(* CODESYS project EZS2_Template.project

Project tree, tasks and I/O mapping:
  Device : Berghof PPC V3 Control, Berghof Automation GmbH, version 3.12.3.0
    application Application
      libraries: Standard, * (System)
      task MainTask (cyclic, interval 4000 µs, priority 16) calls MAIN
      task EtherCAT_Task (cyclic, interval 4000 µs, priority 0) calls EtherCAT_Master.EtherCAT_Task [EtherCAT_Master.EtherCAT_Task]
      global variables Globale_Variablen
      POUs/
        program MAIN [FBD]
        Simulation/
          program SimulationPRG [ST]
          function block SimWerkstueck [SFC]: Init_entry, Einlegestation_active, Band1_active, Uebergabestation1_active, Fraesstation_active, Bohrstation_active, Uebergabestation_active, Ausgabestation_active, Init_active, Init_active_0, Einlegestation_entry
          program Simu [ST]
          function block SimSchieber [ST]
        Steuerung/
          program Steuerung [FBD]
          function block EinAusgabe [SFC]: waitForPstation_entry, bandactive_entry, overshoot_active, overshoot_exit, Init_active, bandactive_active
          function block Uebergabe [SFC]: SationEmty_entry, Push_active, Push_entry, Push_exit, Pull_entry, Pull_active, Pull_exit, StationEmty_exit
      visualisation TAKTSTRASSE
    EtherCAT_Master : EtherCAT Master, 3S - Smart Software Solutions GmbH, version 3.5.8.40
        settings: NetworkName = 'eth1'; NetworkName = "eth1"; SelectNetworkByName = True
      onboard_Buskoppler : onboard Buscoupler, Berghof Automation GmbH, version Revision=16#00000001
          settings: StationAlias = 0; DC sync0 cycletime = 4000; DC sync1 cycletime = 4000
        E_I_O_DI16_DO16 : DI16/DO16 1ms 0.5A (204 800 100), Berghof Automation GmbH, version Revision=16#00000001
            settings: StationAlias = 0; DC sync0 cycletime = 4000; DC sync1 cycletime = 4000
            unmapped channels: DigitalOutput0, DigitalOutput1, DigitalOutput2, DigitalOutput3, DigitalOutput4, DigitalOutput5, DigitalOutput6, DigitalOutput7, DigitalOutput8, DigitalOutput9, DigitalOutput10, DigitalOutput11, DigitalOutput12, DigitalOutput13, DigitalOutput14, DigitalOutput15, DigitalInput0, DigitalInput1, DigitalInput2, DigitalInput3, DigitalInput4, DigitalInput5, DigitalInput6, DigitalInput7, DigitalInput8, DigitalInput9, DigitalInput10, DigitalInput11, DigitalInput12, DigitalInput13, DigitalInput14, DigitalInput15
  libraries: VisuSymbols, 3.5.10.0 (System)
  text list GlobalTextList
*)

// Device/Application/Globale_Variablen
VAR_GLOBAL
(***** STUDENTEN VARIABLEN *****)

	L1:	BOOL;	(* Lichtschranke 1 (Einlegestation) *)
	L2:	BOOL;	(* Lichtschranke 2 (Einlegestation) *)
	L3:	BOOL;	(* Lichtschranke 3 (Fraeser) *)
	L4:	BOOL;	(* Lichtschranke 4 (Bohrer) *)
	L5:	BOOL;	(* Lichtschranke 5 (Ausgabestation) *)
	
	E1:	BOOL;	(* Endtaster 1 (Uebergabestation 1) *)
	E2:	BOOL;	(* Endtaster 2 (Uebergabestation 1) *)
	E3: BOOL;	(* Endtaster 3 (Uebergabestation 2) *)
	E4:	BOOL;	(* Endtaster 4 (Uebergabestation 2) *)
	
	B1	AT %QX0.0:	BOOL;	(* Foerderband 1 (Einlegestation) *)
	B2	AT %QX0.1:	BOOL;	(* Foerderband 2 (Fraeser) *)
	B3	AT %QX0.2:	BOOL;	(* Foerderband 3 (Bohrer) *)
	B4	AT %QX0.3:	BOOL;	(* Foerderband 4 (Ausgabestation) *)
	
	M1	AT %QX0.5:	BOOL;	(* Motor 1 (Uebergabestation 1) *)
	M2	AT %QX0.6:	BOOL;	(* Motor 2 (Fraeser) *)
	M3	AT %QX0.7:	BOOL;	(* Motor 3 (Bohrer) *)
	M4	AT %QX0.8:	BOOL;	(* Motor 4 (Uebergabestation 2) *)
	
	R1	AT %QX0.10:	BOOL;	(* Relais 1 (Uebergabestation 1) *)
	R2	AT %QX0.11:	BOOL;	(* Relais 2 (Uebergabestation 2) *)

(***** ENDE ***** STUDENTEN VARIABLEN *****)

	L1_real	AT %IX0.0:	BOOL;	(* Lichtschranke 1 (Einlegestation) *)
	L2_real	AT %IX0.1:	BOOL;	(* Lichtschranke 2 (Einlegestation) *)
	L3_real	AT %IX0.2:	BOOL;	(* Lichtschranke 3 (Fraeser) *)
	L4_real	AT %IX0.3:	BOOL;	(* Lichtschranke 4 (Bohrer) *)
	L5_real	AT %IX0.4:	BOOL;	(* Lichtschranke 5 (Ausgabestation) *)
	
	E1_real	AT %IX0.6:	BOOL;	(* Endanschlag 1 (Uebergabestation 1) *)
	E2_real	AT %IX0.7:	BOOL;	(* Endanschlag 2 (Uebergabestation 1) *)
	E3_real	AT %IX0.8: 	BOOL;	(* Endanschlag 3 (Uebergabestation 2) *)
	E4_real	AT %IX0.9:	BOOL;	(* Endanschlag 4 (Uebergabestation 2) *)

	SIMULATION: BOOL := TRUE;

END_VAR

// Device/Application/POUs/MAIN
PROGRAM MAIN
VAR
END_VAR

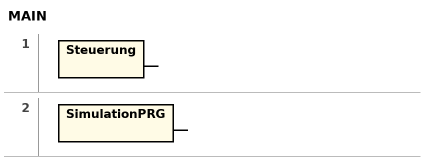
// NETWORK 1
Steuerung();

// NETWORK 2
SimulationPRG();

END_PROGRAM

// Device/Application/POUs/Steuerung/Steuerung
PROGRAM Steuerung
VAR
	Eingabe: EinAusgabe;
	Ue1Emty:BOOL;
	overTimeEin:TIME:=T#2S;
	Uebergabe_1: Uebergabe;
	finishedEin: BOOL;
	toUe1: BOOL;
	toFrae: BOOL;
	Ue1Fin: BOOL;
END_VAR

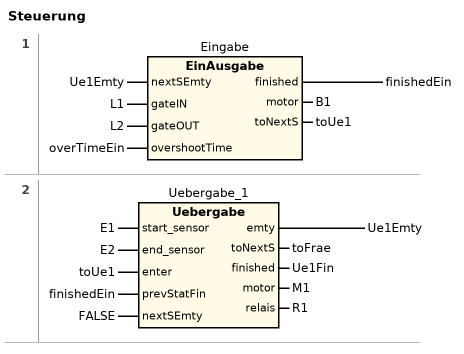
// NETWORK 1
Eingabe(
    nextSEmty := Ue1Emty,
    gateIN := L1,
    gateOUT := L2,
    overshootTime := overTimeEin,
    motor => B1,
    toNextS => toUe1); // EinAusgabe
finishedEin := Eingabe.finished;

// NETWORK 2
Uebergabe_1(
    start_sensor := E1,
    end_sensor := E2,
    enter := toUe1,
    prevStatFin := finishedEin,
    nextSEmty := FALSE,
    toNextS => toFrae,
    finished => Ue1Fin,
    motor => M1,
    relais => R1); // Uebergabe
Ue1Emty := Uebergabe_1.emty;

END_PROGRAM

// Device/Application/POUs/Steuerung/EinAusgabe
FUNCTION_BLOCK EinAusgabe 
VAR_INPUT
	nextSEmty:BOOL;
	gateIN:BOOL;
	gateOUT:BOOL;
	overshootTime:TIME;
END_VAR
VAR_OUTPUT
	finished: BOOL;
	motor:BOOL;
	toNextS: BOOL;
END_VAR
VAR
	timer:	TON;
END_VAR

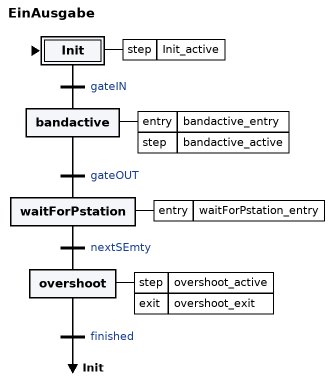
INITIAL_STEP Init:
    Init_active(N);  // step action
END_STEP
TRANSITION FROM Init TO bandactive
    := gateIN;
END_TRANSITION
STEP bandactive:
    bandactive_entry(P1);  // entry action
    bandactive_active(N);  // step action
END_STEP
TRANSITION FROM bandactive TO waitForPstation
    := gateOUT;
END_TRANSITION
STEP waitForPstation:
    waitForPstation_entry(P1);  // entry action
END_STEP
TRANSITION FROM waitForPstation TO overshoot
    := nextSEmty;
END_TRANSITION
STEP overshoot:
    overshoot_active(N);  // step action
    overshoot_exit(P0);  // exit action
END_STEP
TRANSITION FROM overshoot TO Init
    := finished;
END_TRANSITION

ACTION waitForPstation_entry:
motor:=FALSE;
END_ACTION

ACTION bandactive_entry:
motor:=true;
END_ACTION

ACTION overshoot_active:
timer(IN:=TRUE,PT:=overshootTime);
finished:=timer.Q;
toNextS:=TRUE;
motor:=True;
END_ACTION

ACTION overshoot_exit:
timer(IN:=FALSE);
motor:=FALSE;
toNextS:=false;
END_ACTION

ACTION Init_active:
timer(IN:=FALSE);
motor:=false;
END_ACTION

ACTION bandactive_active:
motor:=true;
END_ACTION

END_FUNCTION_BLOCK

// Device/Application/POUs/Steuerung/Uebergabe
FUNCTION_BLOCK Uebergabe
VAR_INPUT
	start_sensor: BOOL;		(* Wert des ersten Sensors - Schieber ist eingefahren *)
	end_sensor: BOOL;		(* Motor des Schiebers *)
	enter:BOOL;
	prevStatFin:BOOL;
	nextSEmty:BOOL;	 
END_VAR
VAR_OUTPUT
	emty:BOOL;
	toNextS:BOOL;
	finished:BOOL;
	motor: BOOL;
	relais: BOOL;
END_VAR
VAR
END_VAR

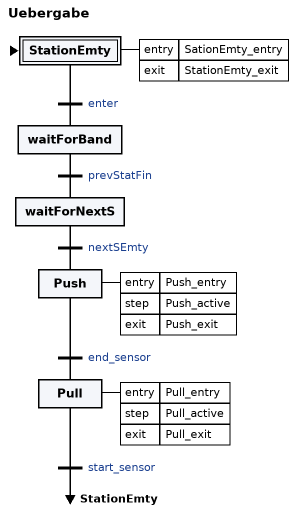
INITIAL_STEP StationEmty:
    SationEmty_entry(P1);  // entry action
    StationEmty_exit(P0);  // exit action
END_STEP
TRANSITION FROM StationEmty TO waitForBand
    := enter;
END_TRANSITION
STEP waitForBand:
END_STEP
TRANSITION FROM waitForBand TO waitForNextS
    := prevStatFin;
END_TRANSITION
STEP waitForNextS:
END_STEP
TRANSITION FROM waitForNextS TO Push
    := nextSEmty;
END_TRANSITION
STEP Push:
    Push_entry(P1);  // entry action
    Push_active(N);  // step action
    Push_exit(P0);  // exit action
END_STEP
TRANSITION FROM Push TO Pull
    := end_sensor;
END_TRANSITION
STEP Pull:
    Pull_entry(P1);  // entry action
    Pull_active(N);  // step action
    Pull_exit(P0);  // exit action
END_STEP
TRANSITION FROM Pull TO StationEmty
    := start_sensor;
END_TRANSITION

ACTION SationEmty_entry:
emty:=TRUE;
motor:=FALSE;
finished:=FALSE;
toNextS:=FALSE;
END_ACTION

ACTION Push_active:

motor:=true;
END_ACTION

ACTION Push_entry:
relais:=FALSE;
toNextS:=True;
END_ACTION

ACTION Push_exit:
motor:=FALSE;
finished:=TRUE;
END_ACTION

ACTION Pull_entry:
relais:=TRUE;
END_ACTION

ACTION Pull_active:
motor:=TRUE;
END_ACTION

ACTION Pull_exit:
motor:=false;
END_ACTION

ACTION StationEmty_exit:
emty:=false;
END_ACTION

END_FUNCTION_BLOCK

// Device/Application/POUs/Simulation/SimulationPRG
PROGRAM SimulationPRG
VAR
END_VAR

(* DO NOT CHANGE *)
IF (NOT SIMULATION) THEN
	L1 := L1_real;	(* Lichtschranke 1 (Einlegestation) *)	
	L2 := L2_real;	(* Lichtschranke 2 (Einlegestation) *)
	L3 := L3_real;	(* Lichtschranke 3 (Fraeser) *)
	L4 := L4_real;	(* Lichtschranke 4 (Bohrer) *)
	L5 := L5_real;	(* Lichtschranke 5 (Ausgabestation) *)
	
	E1 := E1_real;	(* Endtaster 1 (Uebergabestation 1) *)
	E2 := E2_real;	(* Endtaster 2 (Uebergabestation 1) *)
	E3 := E3_real;	(* Endtaster 3 (Uebergabestation 2) *)
	E4 := E4_real;	(* Endtaster 4 (Uebergabestation 2) *)
ELSE
	Simu(); 
END_IF

END_PROGRAM

// Device/Application/POUs/Simulation/Simu
PROGRAM Simu
VAR
	schieber1: SimSchieber; 	(* Simulationsbaustein für den ersten Schieber *)
	schieber2: SimSchieber;		(* Simulationsbaustein für den zweiten Schieber *)
	token1: SimWerkstueck;		(* Simulationsbaustein für das erste Werkstück *)
	token2: SimWerkstueck; 		(* Simulationsbaustein für das zweite Werkstück *) 
END_VAR

(* Aufruf des ersten Schiebers *) 
schieber1(start_pos := 0, end_pos := 40, motor := M1, relais := R1); 
E1 := schieber1.start_sensor;
E2 := schieber1.end_sensor;

(* Aufruf des zweiten Schiebers *)
schieber2(start_pos := 0, end_pos := 40, motor := M4, relais := R2); 
E3 := schieber2.start_sensor;
E4 := schieber2.end_sensor;

(* TODO: Aufruf der Werkstücke *)
token1(schieber1_pos:=schieber1.pos,schieber2_pos:=schieber2.pos);
token2(schieber1_pos:=schieber1.pos,schieber2_pos:=schieber2.pos);

(* TODO: Zuweisung für die Lichtschranken *) 
L1:=token1.L1_token OR token2.L1_token ;
L2:=token1.L2_token OR token2.L2_token ;
L3:=token1.L3_token OR token2.L3_token ;
L4:=token1.L4_token OR token2.L4_token ;
L5:=token1.L5_token OR token2.L5_token ;

END_PROGRAM

// Device/Application/POUs/Simulation/SimSchieber
FUNCTION_BLOCK SimSchieber
VAR_INPUT
	start_pos: INT;		(* Position, wenn der Schieber eingefahren ist *)
	end_pos: INT;		(* Position, wenn der Schieber ausgefahren ist *) 
	motor: BOOL;		(* Motor des Schiebers *)
	relais: BOOL;		(* Relais des Schiebers *) 
END_VAR
VAR_OUTPUT
	pos: INT := start_pos;	(* Aktuelle Position des Schiebers *)
	start_sensor: BOOL;		(* Wert des ersten Sensors - Schieber ist eingefahren *)
	end_sensor: BOOL; 		(* Wert des zweiten Sensors - Schieber ist ausgefahren *) 
END_VAR

(* TODO: (Rück-)Setzen der virtuellen Sensoren start_sensor und end_sensor *) 
IF pos=end_pos THEN
	end_sensor:=TRUE;
ELSE
	end_sensor:=FALSE;	
END_IF
IF pos=start_pos THEN
	start_sensor:=TRUE;
ELSE
	start_sensor:=FALSE;
END_IF
IF NOT relais AND motor AND NOT end_sensor THEN
	pos:=pos+1;
ELSIF relais AND motor AND NOT start_sensor THEN
	pos:=pos-1;
END_IF

(* TODO: Aktualisiere (inkrementiere oder dekrementiere) die aktuelle Position des Schiebers *)

END_FUNCTION_BLOCK

// Device/Application/POUs/Simulation/SimWerkstueck
FUNCTION_BLOCK SimWerkstueck
VAR_INPUT
	start: BOOL := FALSE;	(* Wird  voon der Visualisierung gesetzt, wenn das Werkstück auf das Band gelegt wird *)
	schieber1_pos: INT;		(* Aktuelle Position des ersten Schiebers *)
	schieber2_pos: INT; 	(* Aktuelle Position des zweiten Schiebers *)
END_VAR
VAR_OUTPUT
	pos_x: INT;				(* X Position des Werkstücks relativ zum Startpunkt *) 
	pos_y: INT; 			(* Y Position des Werkstücks relativ zum Startpunkt *)
	visible: BOOL;			(* True, falls das Werkstück in der Anlage ist *) 
	L1_token: BOOL;			(* True, falls das Werkstück vor der 1. Lichtschranke ist *) 
	L2_token: BOOL;			(* True, falls das Werkstück vor der 2. Lichtschranke ist *) 
	L3_token: BOOL;			(* True, falls das Werkstück vor der 3. Lichtschranke ist *) 
	L4_token: BOOL;			(* True, falls das Werkstück vor der 4. Lichtschranke ist *) 
	L5_token: BOOL; 		(* True, falls das Werkstück vor der 5. Lichtschranke ist *) 
END_VAR
VAR
	toStation2: BOOL;
	toFraesStation: BOOL;
	toBohrstation: BOOL;
	toUestation2: BOOL;
	toAusgabestation: BOOL;
	toEnd: BOOL;
END_VAR

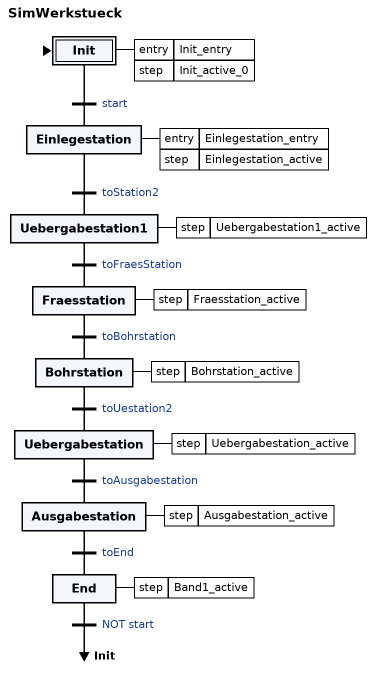
INITIAL_STEP Init:
    Init_entry(P1);  // entry action
    Init_active_0(N);  // step action
END_STEP
TRANSITION FROM Init TO Einlegestation
    := start;
END_TRANSITION
STEP Einlegestation:
    Einlegestation_entry(P1);  // entry action
    Einlegestation_active(N);  // step action
END_STEP
TRANSITION FROM Einlegestation TO Uebergabestation1
    := toStation2;
END_TRANSITION
STEP Uebergabestation1:
    Uebergabestation1_active(N);  // step action
END_STEP
TRANSITION FROM Uebergabestation1 TO Fraesstation
    := toFraesStation;
END_TRANSITION
STEP Fraesstation:
    Fraesstation_active(N);  // step action
END_STEP
TRANSITION FROM Fraesstation TO Bohrstation
    := toBohrstation;
END_TRANSITION
STEP Bohrstation:
    Bohrstation_active(N);  // step action
END_STEP
TRANSITION FROM Bohrstation TO Uebergabestation
    := toUestation2;
END_TRANSITION
STEP Uebergabestation:
    Uebergabestation_active(N);  // step action
END_STEP
TRANSITION FROM Uebergabestation TO Ausgabestation
    := toAusgabestation;
END_TRANSITION
STEP Ausgabestation:
    Ausgabestation_active(N);  // step action
END_STEP
TRANSITION FROM Ausgabestation TO End
    := toEnd;
END_TRANSITION
STEP End:
    Band1_active(N);  // step action
END_STEP
TRANSITION FROM End TO Init
    := NOT start;
END_TRANSITION

ACTION Init_entry:
pos_x := 0;
pos_y := 0; 
visible := FALSE;
L1_token := FALSE;
L2_token := FALSE;
L3_token := FALSE;
L4_token := FALSE;
L5_token := FALSE;
toStation2:=FALSE;
toFraesStation:=FALSE;
toBohrstation:=FALSE;
toUestation2:=FALSE;
toAusgabestation:=FALSE;
toEnd:=FALSE;
END_ACTION

ACTION Einlegestation_active:
IF pos_y>=-20 AND pos_x=0 THEN
	L1_token:=TRUE;
ELSE
	L1_token:=FALSE;
END_IF
IF pos_y<=-50 AND pos_y>=-90 AND pos_x=0 THEN
	L2_token:=TRUE;
ELSE
	L2_token:=FALSE;
END_IF
IF B1 THEN
	pos_y:=pos_y-1;
END_IF
IF pos_y=-110 THEN
	toStation2:=TRUE;
END_IF
END_ACTION

ACTION Band1_active:
visible:=FALSE;
start:=FALSE;
END_ACTION

ACTION Uebergabestation1_active:
IF NOT R1 THEN
	pos_x:=schieber1_pos;
END_IF
IF pos_x>=40 THEN
	toFraesStation:=TRUE;
END_IF
END_ACTION

ACTION Fraesstation_active:
IF pos_y=-110 AND pos_x>=100 AND pos_x<=140 THEN
	L3_token:=TRUE;
ELSE
	L3_token:=FALSE;
END_IF
IF B2 THEN
	pos_x:=pos_x+1;
END_IF
IF pos_x=150 THEN
	toBohrstation:=TRUE;
END_IF
END_ACTION

ACTION Bohrstation_active:
IF pos_y=-110 AND pos_x>=210 AND pos_x<=250 AND visible THEN
	L4_token:=TRUE;
ELSE
	L4_token:=FALSE;
END_IF
IF B3 THEN
	pos_x:=pos_x+1;
END_IF
IF pos_x=270 THEN
	toUestation2:=TRUE;
END_IF
END_ACTION

ACTION Uebergabestation_active:
IF NOT R2 THEN
	pos_y:=schieber2_pos-110;
END_IF
IF pos_y>=-70 THEN
	toausgabestation:=TRUE;
END_IF
END_ACTION

ACTION Ausgabestation_active:
IF pos_y<=0 AND pos_y>=-40 AND pos_x=270 THEN
	L5_token:=TRUE;
ELSE
	L5_token:=FALSE;
END_IF
IF B4 THEN
	pos_y:=pos_y+1;
END_IF
IF pos_y=0 THEN
	toEnd:=TRUE;
END_IF
END_ACTION

ACTION Init_active:
pos_x:=0;
pos_y:=0;
visible:=TRUE;
start:=TRUE;
END_ACTION

ACTION Init_active_0:

END_ACTION

ACTION Einlegestation_entry:
visible := TRUE;
END_ACTION

END_FUNCTION_BLOCK

// Device/Application/TAKTSTRASSE
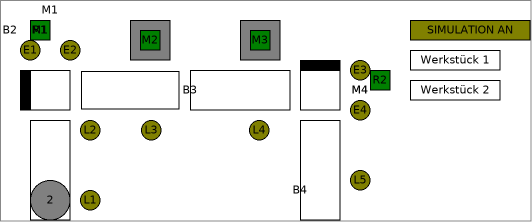
VISUALIZATION TAKTSTRASSE  // 532x222
    Rectangle (30,120 40x100)
    Rectangle (300,70 40x40)
    Rectangle (30,70 40x40)
    RoundedRectangle (30,20 20x20), "R1", colour toggle: Globale_Variablen.R1, input disabled if: (NOT SIMULATION) <> 0
        toggle Globale_Variablen.R1
    RoundedRectangle (370,70 20x20), "R2", colour toggle: R2, input disabled if: NOT SIMULATION
        toggle R2
    RoundedRectangle (410,50 90x20), "Werkstück 1", colour toggle: Simu.token1.visible, invisible if: NOT SIMULATION
        toggle Simu.token1.start
    RoundedRectangle (410,20 120x20), "SIMULATION AN", colour toggle: Globale_Variablen.SIMULATION
        toggle Globale_Variablen.SIMULATION
    Polygon (40,30), "M1", colour toggle: Globale_Variablen.M1, invisible if: Globale_Variablen.R1, input disabled if: (NOT SIMULATION) <> 0
        toggle Globale_Variablen.M1
    Polygon (50,10), "M1", colour toggle: Globale_Variablen.M1, invisible if: (NOT R1) <> 0, input disabled if: (NOT SIMULATION) <> 0
        toggle Globale_Variablen.M1
    Polygon (360,90), "M4", colour toggle: M4, invisible if: R2, input disabled if: NOT SIMULATION
        toggle M4
    Polygon (360,90), "M4", colour toggle: M4, invisible if: NOT R2, input disabled if: NOT SIMULATION
        toggle M4
    Rectangle (81,71 98x38)
    Polygon (10,30), "B2", colour toggle: B2, input disabled if: NOT SIMULATION
        toggle B2
    Rectangle (190,70 100x40)
    Polygon (190,90), "B3", colour toggle: B3, input disabled if: NOT SIMULATION
        toggle B3
    Ellipse (141,120 20x20), "L3", colour toggle: L3, input disabled if: NOT SIMULATION
        toggle L3
    Polyline (140,50)
    Ellipse (249,120 20x20), "L4", colour toggle: L4, input disabled if: NOT SIMULATION
        toggle L4
    Polyline (250,50)
    Ellipse (20,40 20x20), "E1", colour toggle: E1, input disabled if: NOT SIMULATION
        toggle E1
    Polygon (30,50)
    Ellipse (60,40 20x20), "E2", colour toggle: E2, input disabled if: NOT SIMULATION
        toggle E2
    Polygon (70,50)
    RoundedRectangle (130,20 40x40)
    RoundedRectangle (140,30 20x20), "M2", colour toggle: M2, input disabled if: NOT SIMULATION
        toggle M2
    RoundedRectangle (240,20 40x40)
    RoundedRectangle (250,30 20x20), "M3", colour toggle: M3, input disabled if: NOT SIMULATION
        toggle M3
    Ellipse (350,60 20x20), "E3", colour toggle: E3, input disabled if: NOT SIMULATION
        toggle E3
    Polygon (340,70)
    Ellipse (350,100 20x20), "E4", colour toggle: E4, input disabled if: NOT SIMULATION
        toggle E4
    Polygon (340,110)
    Ellipse (350,170 20x20), "L5", colour toggle: L5, input disabled if: NOT SIMULATION
        toggle L5
    Ellipse (80,190 20x20), "L1", colour toggle: L1, input disabled if: NOT SIMULATION
        toggle L1
    Polygon (50,200), "B1", colour toggle: B1, input disabled if: NOT SIMULATION
        toggle B1
    Polyline (70,190)
    Ellipse (80,120 20x20), "L2", colour toggle: L2, input disabled if: NOT SIMULATION
        toggle L2
    Polyline (70,130)
    Rectangle (300,120 40x100)
    Polygon (300,190), "B4", colour toggle: B4, input disabled if: NOT SIMULATION
        toggle B4
    Polyline (340,190)
    Ellipse (30,180 40x40), "1", invisible if: NOT Simu.token1.visible
        p3560616238: Simu.token1.pos_x
        p2738717112: Simu.token1.pos_y
    Rectangle (20,70 10x40)
        p3560616238: Simu.schieber1.pos
    Rectangle (300,60 40x10)
        p2738717112: Simu.schieber2.pos
    RoundedRectangle (410,80 90x20), "Werkstück 2", colour toggle: Simu.token2.visible, invisible if: NOT SIMULATION
        toggle Simu.token2.start
    Ellipse (30,180 40x40), "2", invisible if: NOT Simu.token2.visible
        p3560616238: Simu.token2.pos_x
        p2738717112: Simu.token2.pos_y
END_VISUALIZATION
